// Block: CarriageLub_PERS

DATA_BLOCK CarriageLub_PERS
VERSION : 0.1
   NON_RETAIN
   VAR
      Carriage_SlideLubr : Struct
         Control : LubrValve_Pers;
         EvLub : LubrPump_Par;
      END_STRUCT;
      CarriageLub_Pers_HMI_ResetCounter : Bool;
   END_VAR

BEGIN
   // No initialization required
END_DATA_BLOCK
